PROGRAM P_AxisControl
VAR
END_VAR

//Axis Control program based on youtube series Twincat 3 NC Videos MB05a until MB17b plus MB22 by @electricalautomation https://www.youtube.com/watch?v=BxRAOdTks9I&list=PL762SfoJC-e8NbAUQ-H7a_TOdqrlBPCw4&index=25

AXIS1_LD();

GVL_AXIS1.bBC_ResetExe := G_Inputs.bJoystickLeftEnable OR G_Inputs.bAutoModeSelector;

GVL_AXIS1.EnuMoveVelDirection := G_Sensors.MCDirectionAxis1;

GVL_AXIS1.bBC_PowerEnCmd := G_Inputs.bManualModeSelector OR G_Inputs.bAutoModeSelector;
GVL_AXIS1.bBC_PowerEnNegative := G_Inputs.bManualModeSelector OR G_Inputs.bAutoModeSelector;
GVL_AXIS1.bBC_PowerEnPositive := G_Inputs.bManualModeSelector OR G_Inputs.bAutoModeSelector;

GVL_AXIS1.lrBC_JogVelocity := 100;
GVL_AXIS1.lrBC_PowerOverride := 50;

GVL_AXIS1.lrBC_MoveAbsPosition := GVL_InverseKinematics.fStrokeActuatorMainInverse*1000; //Position in mm

// Jog control

(*
IF G_Sensors.fJoystickLeftNormalizedX  > 0 AND G_Inputs.bJoystickLeftEnable THEN
	GVL_AXIS1.bBC_JogRev := TRUE;
ELSIF G_Sensors.fJoystickLeftNormalizedX < 0 AND G_Inputs.bJoystickLeftEnable THEN
	GVL_AXIS1.bBC_JogFwd := TRUE;
ELSE
	 GVL_AXIS1.bBC_JogFwd := FALSE;
	 GVL_AXIS1.bBC_JogRev := FALSE;
END_IF

*)



// Manual velocity control
IF G_Sensors.fJoystickLeftNormalizedX  > 0 AND G_Inputs.bJoystickLeftEnable AND G_Inputs.bManualModeSelector THEN
	GVL_AXIS1.lrBC_PowerOverride := ABS(G_Sensors.fJoystickLeftNormalizedX) * 100;
	GVL_AXIS1.stBC_VelCmd.EnuDirection := MC_Positive_Direction;
	GVL_AXIS1.stBC_VelCmd.bExe := TRUE;
ELSIF G_Sensors.fJoystickLeftNormalizedX < 0 AND G_Inputs.bJoystickLeftEnable AND G_Inputs.bManualModeSelector THEN
	GVL_AXIS1.lrBC_PowerOverride := ABS(G_Sensors.fJoystickLeftNormalizedX) * 100;
	GVL_AXIS1.stBC_VelCmd.EnuDirection := MC_Negative_Direction;
	GVL_AXIS1.stBC_VelCmd.bExe := TRUE;
ELSIF G_Inputs.bAutoModeSelector THEN
	GVL_AXIS1.lrBC_PowerOverride := 10;
	//GVL_AXIS1.stBC_VelCmd.EnuDirection := MC_Positive_Direction;
	GVL_AXIS1.stBC_VelCmd.bExe := TRUE;
	GVL_AXIS1.bBC_MoveAbsExe := TRUE;
ELSE
	 GVL_AXIS1.lrBC_PowerOverride := 0;
	 //GVL_AXIS1.stBC_VelCmd.EnuDirection := MC_Current_Direction;
	 GVL_AXIS1.stBC_VelCmd.bExe := FALSE;
END_IF


// Automatic position control

IF G_Inputs.bAutoModeSelector THEN
	GVL_AXIS1.lrBC_PowerOverride := 10;
	//GVL_AXIS1.stBC_VelCmd.EnuDirection := MC_Positive_Direction;
	GVL_AXIS1.stBC_VelCmd.bExe := TRUE;
	GVL_AXIS1.bBC_MoveAbsExe := TRUE;
ELSE
	 GVL_AXIS1.lrBC_PowerOverride := 0;
	 //GVL_AXIS1.stBC_VelCmd.EnuDirection := MC_Current_Direction;
	 GVL_AXIS1.stBC_VelCmd.bExe := FALSE;
END_IF


AXIS2_LD();

GVL_AXIS2.bSJ_ResetExe := G_Inputs.bJoystickRightEnable;

GVL_AXIS2.EnuMoveVelDirection := G_Sensors.MCDirectionAxis2;

GVL_AXIS2.bSJ_PowerEnCmd := G_Inputs.bManualModeSelector;
GVL_AXIS2.bSJ_PowerEnNegative := G_Inputs.bManualModeSelector;
GVL_AXIS2.bSJ_PowerEnPositive := G_Inputs.bManualModeSelector;

GVL_AXIS2.lrSJ_JogVelocity := 100;


// Velocity control
IF G_Sensors.fJoystickRightNormalizedX  > 0 AND G_Inputs.bJoystickRightEnable THEN
	GVL_AXIS2.lrSJ_PowerOverride := ABS(G_Sensors.fJoystickRightNormalizedX) * 100;
	GVL_AXIS2.stSJ_VelCmd.EnuDirection := MC_Positive_Direction;
	GVL_AXIS2.stSJ_VelCmd.bExe := TRUE;
ELSIF G_Sensors.fJoystickRightNormalizedX < 0 AND G_Inputs.bJoystickRightEnable THEN
	GVL_AXIS2.lrSJ_PowerOverride := ABS(G_Sensors.fJoystickRightNormalizedX) * 100;
	GVL_AXIS2.stSJ_VelCmd.EnuDirection := MC_Negative_Direction;
	GVL_AXIS2.stSJ_VelCmd.bExe := TRUE;
ELSE
	 GVL_AXIS2.lrSJ_PowerOverride := 0;
	 //GVL_AXIS2.stSJ_VelCmd.EnuDirection := MC_Current_Direction;
	 GVL_AXIS2.stSJ_VelCmd.bExe := FALSE;
END_IF


AXIS3_LD();

GVL_AXIS3.bTC_ResetExe := G_Inputs.bJoystickLeftEnable;

GVL_AXIS3.EnuMoveVelDirection := G_Sensors.MCDirectionAxis3;

GVL_AXIS3.bTC_PowerEnCmd := G_Inputs.bManualModeSelector;
GVL_AXIS3.bTC_PowerEnNegative := G_Inputs.bManualModeSelector;
GVL_AXIS3.bTC_PowerEnPositive := G_Inputs.bManualModeSelector;

GVL_AXIS3.lrTC_JogVelocity := 100;


// Velocity control
IF G_Sensors.fJoystickLeftNormalizedY  > 0 AND G_Inputs.bJoystickLeftEnable THEN
	GVL_AXIS3.lrTC_PowerOverride := ABS(G_Sensors.fJoystickLeftNormalizedY) * 100;
	GVL_AXIS3.stTC_VelCmd.EnuDirection := MC_Positive_Direction;
	GVL_AXIS3.stTC_VelCmd.bExe := TRUE;
ELSIF G_Sensors.fJoystickLeftNormalizedY < 0 AND G_Inputs.bJoystickLeftEnable THEN
	GVL_AXIS3.lrTC_PowerOverride := ABS(G_Sensors.fJoystickLeftNormalizedY) * 100;
	GVL_AXIS3.stTC_VelCmd.EnuDirection := MC_Negative_Direction;
	GVL_AXIS3.stTC_VelCmd.bExe := TRUE;
ELSE
	 GVL_AXIS3.lrTC_PowerOverride := 0;
	 //GVL_AXIS3.stTC_VelCmd.EnuDirection := MC_Current_Direction;
	 GVL_AXIS3.stTC_VelCmd.bExe := FALSE;
END_IF

(*
AXIS4_LD();

//Safety
GVL_Safety_AXIS4.bSafetyRestart := GVL_AXIS4.bInAckSignal;
GVL_Safety_AXIS4.bErrorAck		:= GVL_AXIS4.bInAckSignal;
GVL_Safety_AXIS4.bSafetyRun		:= TRUE;

//
GVL_AXIS4.bWM_ResetExe := G_Inputs.bJoystickLeftEnable;

GVL_AXIS4.EnuMoveVelDirection := G_Sensors.MCDirectionAxis4;

GVL_AXIS4.bWM_PowerEnCmd := G_Inputs.bManualModeSelector;
GVL_AXIS4.bWM_PowerEnNegative := G_Inputs.bManualModeSelector;
GVL_AXIS4.bWM_PowerEnPositive := G_Inputs.bManualModeSelector;

GVL_AXIS4.lrWM_JogVelocity := 100;
//GVL_AXIS4.lrWM_PowerOverride := 50;


// Velocity control
IF G_Sensors.fJoystickLeftNormalizedY  > 0 AND G_Inputs.bJoystickLeftEnable THEN
	GVL_AXIS4.lrWM_PowerOverride := ABS(G_Sensors.fJoystickLeftNormalizedY) * 100;
	GVL_AXIS4.stWM_VelCmd.EnuDirection := MC_Positive_Direction;
	GVL_AXIS4.stWM_VelCmd.bExe := TRUE;
ELSIF G_Sensors.fJoystickLeftNormalizedY < 0 AND G_Inputs.bJoystickLeftEnable THEN
	GVL_AXIS4.lrWM_PowerOverride := ABS(G_Sensors.fJoystickLeftNormalizedY) * 100;
	GVL_AXIS4.stWM_VelCmd.EnuDirection := MC_Negative_Direction;
	GVL_AXIS4.stWM_VelCmd.bExe := TRUE;
ELSE
	 GVL_AXIS4.lrWM_PowerOverride := 0;
	 GVL_AXIS4.stWM_VelCmd.EnuDirection := MC_Current_Direction;
	 GVL_AXIS4.stWM_VelCmd.bExe := FALSE;
END_IF
*)

METHOD AXIS1_LD : BOOL
VAR_INPUT
END_VAR
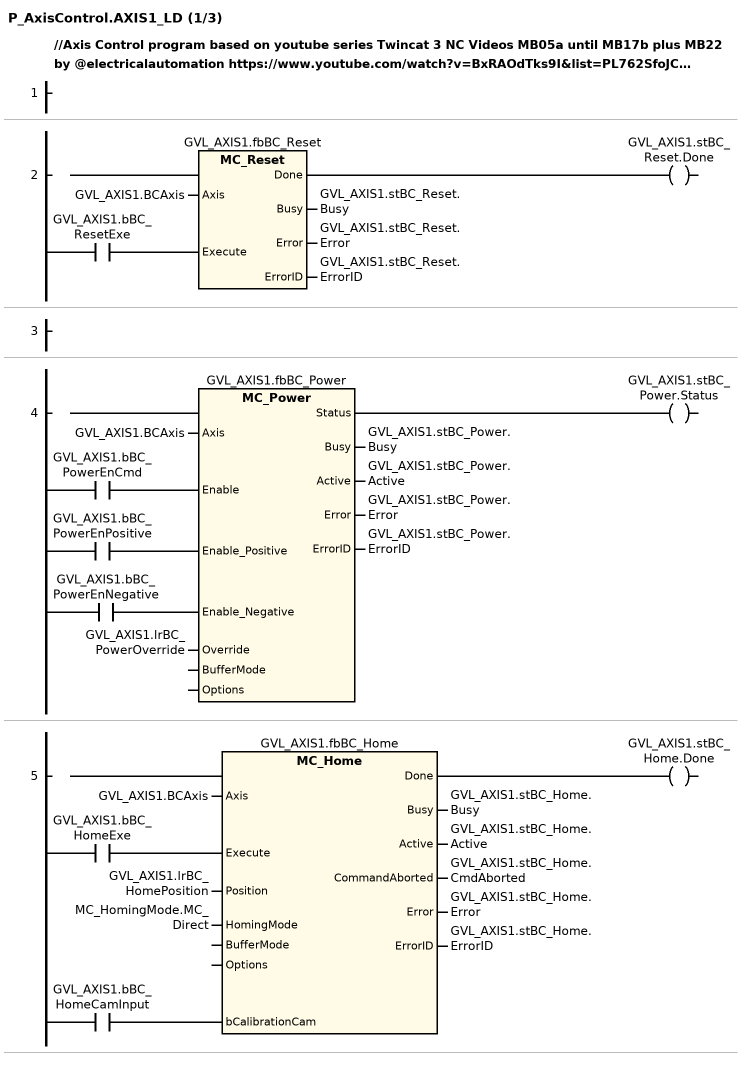
// NETWORK 1: //Axis Control program based on youtube series Twincat 3 NC Videos MB05a until MB17b plus MB22 by @electricalautomation https://www.youtube.com/watch?v=BxRAOdTks9I&list=PL762SfoJC-e8NbAUQ-H7a_TOdqrlBPCw4&index=25

// NETWORK 2
GVL_AXIS1.fbBC_Reset(
    Axis := GVL_AXIS1.BCAxis,
    Execute := GVL_AXIS1.bBC_ResetExe,
    Busy => GVL_AXIS1.stBC_Reset.Busy,
    Error => GVL_AXIS1.stBC_Reset.Error,
    ErrorID => GVL_AXIS1.stBC_Reset.ErrorID); // MC_Reset
GVL_AXIS1.stBC_Reset.Done := GVL_AXIS1.fbBC_Reset.Done;

// NETWORK 3

// NETWORK 4
GVL_AXIS1.fbBC_Power(
    Axis := GVL_AXIS1.BCAxis,
    Enable := GVL_AXIS1.bBC_PowerEnCmd,
    Enable_Positive := GVL_AXIS1.bBC_PowerEnPositive,
    Enable_Negative := GVL_AXIS1.bBC_PowerEnNegative,
    Override := GVL_AXIS1.lrBC_PowerOverride,
    Busy => GVL_AXIS1.stBC_Power.Busy,
    Active => GVL_AXIS1.stBC_Power.Active,
    Error => GVL_AXIS1.stBC_Power.Error,
    ErrorID => GVL_AXIS1.stBC_Power.ErrorID); // MC_Power
GVL_AXIS1.stBC_Power.Status := GVL_AXIS1.fbBC_Power.Status;

// NETWORK 5
GVL_AXIS1.fbBC_Home(
    Axis := GVL_AXIS1.BCAxis,
    Execute := GVL_AXIS1.bBC_HomeExe,
    Position := GVL_AXIS1.lrBC_HomePosition,
    HomingMode := MC_HomingMode.MC_Direct,
    bCalibrationCam := GVL_AXIS1.bBC_HomeCamInput,
    Busy => GVL_AXIS1.stBC_Home.Busy,
    Active => GVL_AXIS1.stBC_Home.Active,
    CommandAborted => GVL_AXIS1.stBC_Home.CmdAborted,
    Error => GVL_AXIS1.stBC_Home.Error,
    ErrorID => GVL_AXIS1.stBC_Home.ErrorID); // MC_Home
GVL_AXIS1.stBC_Home.Done := GVL_AXIS1.fbBC_Home.Done;

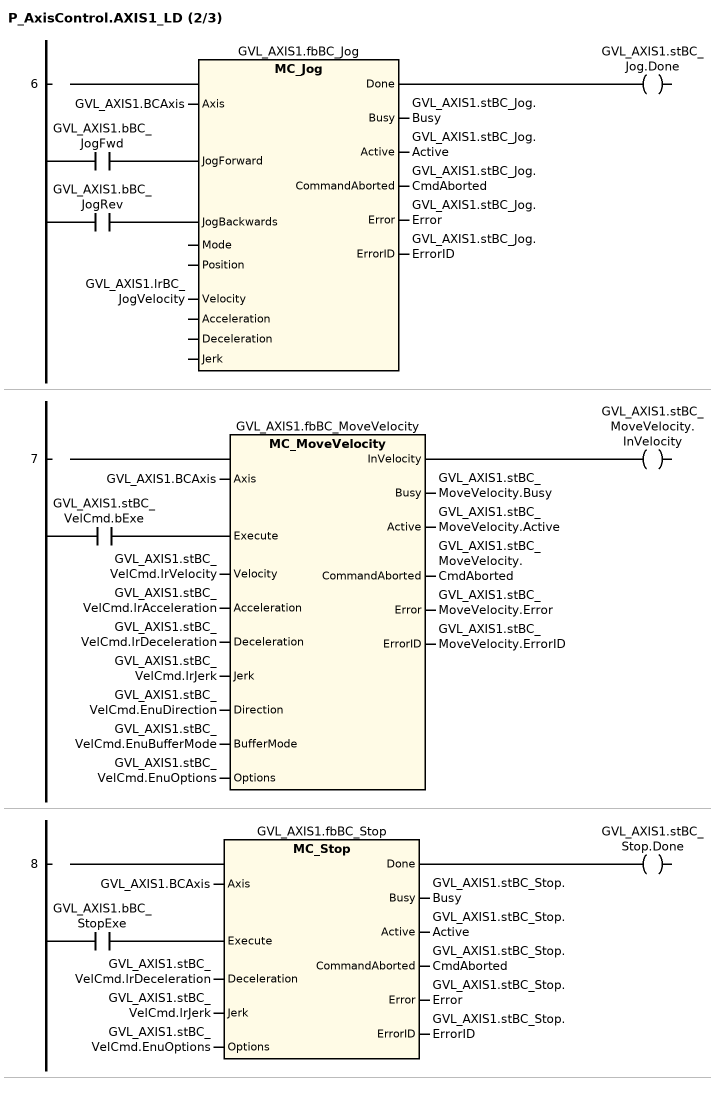
// NETWORK 6
GVL_AXIS1.fbBC_Jog(
    Axis := GVL_AXIS1.BCAxis,
    JogForward := GVL_AXIS1.bBC_JogFwd,
    JogBackwards := GVL_AXIS1.bBC_JogRev,
    Velocity := GVL_AXIS1.lrBC_JogVelocity,
    Busy => GVL_AXIS1.stBC_Jog.Busy,
    Active => GVL_AXIS1.stBC_Jog.Active,
    CommandAborted => GVL_AXIS1.stBC_Jog.CmdAborted,
    Error => GVL_AXIS1.stBC_Jog.Error,
    ErrorID => GVL_AXIS1.stBC_Jog.ErrorID); // MC_Jog
GVL_AXIS1.stBC_Jog.Done := GVL_AXIS1.fbBC_Jog.Done;

// NETWORK 7
GVL_AXIS1.fbBC_MoveVelocity(
    Axis := GVL_AXIS1.BCAxis,
    Execute := GVL_AXIS1.stBC_VelCmd.bExe,
    Velocity := GVL_AXIS1.stBC_VelCmd.lrVelocity,
    Acceleration := GVL_AXIS1.stBC_VelCmd.lrAcceleration,
    Deceleration := GVL_AXIS1.stBC_VelCmd.lrDeceleration,
    Jerk := GVL_AXIS1.stBC_VelCmd.lrJerk,
    Direction := GVL_AXIS1.stBC_VelCmd.EnuDirection,
    BufferMode := GVL_AXIS1.stBC_VelCmd.EnuBufferMode,
    Options := GVL_AXIS1.stBC_VelCmd.EnuOptions,
    Busy => GVL_AXIS1.stBC_MoveVelocity.Busy,
    Active => GVL_AXIS1.stBC_MoveVelocity.Active,
    CommandAborted => GVL_AXIS1.stBC_MoveVelocity.CmdAborted,
    Error => GVL_AXIS1.stBC_MoveVelocity.Error,
    ErrorID => GVL_AXIS1.stBC_MoveVelocity.ErrorID); // MC_MoveVelocity
GVL_AXIS1.stBC_MoveVelocity.InVelocity := GVL_AXIS1.fbBC_MoveVelocity.InVelocity;

// NETWORK 8
GVL_AXIS1.fbBC_Stop(
    Axis := GVL_AXIS1.BCAxis,
    Execute := GVL_AXIS1.bBC_StopExe,
    Deceleration := GVL_AXIS1.stBC_VelCmd.lrDeceleration,
    Jerk := GVL_AXIS1.stBC_VelCmd.lrJerk,
    Options := GVL_AXIS1.stBC_VelCmd.EnuOptions,
    Busy => GVL_AXIS1.stBC_Stop.Busy,
    Active => GVL_AXIS1.stBC_Stop.Active,
    CommandAborted => GVL_AXIS1.stBC_Stop.CmdAborted,
    Error => GVL_AXIS1.stBC_Stop.Error,
    ErrorID => GVL_AXIS1.stBC_Stop.ErrorID); // MC_Stop
GVL_AXIS1.stBC_Stop.Done := GVL_AXIS1.fbBC_Stop.Done;

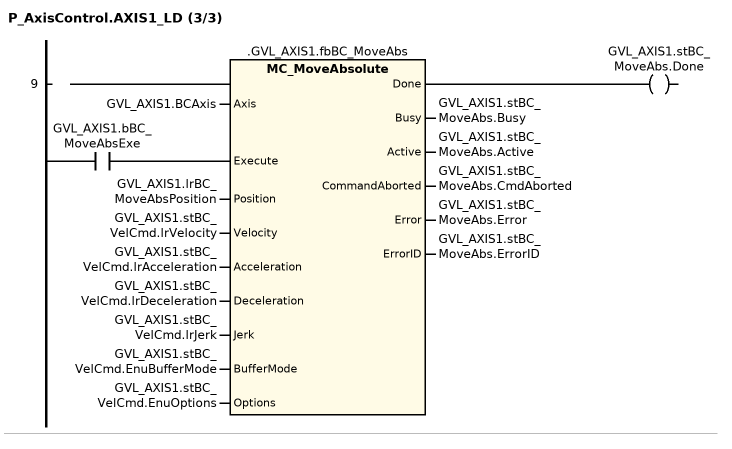
// NETWORK 9
.GVL_AXIS1.fbBC_MoveAbs(
    Axis := GVL_AXIS1.BCAxis,
    Execute := GVL_AXIS1.bBC_MoveAbsExe,
    Position := GVL_AXIS1.lrBC_MoveAbsPosition,
    Velocity := GVL_AXIS1.stBC_VelCmd.lrVelocity,
    Acceleration := GVL_AXIS1.stBC_VelCmd.lrAcceleration,
    Deceleration := GVL_AXIS1.stBC_VelCmd.lrDeceleration,
    Jerk := GVL_AXIS1.stBC_VelCmd.lrJerk,
    BufferMode := GVL_AXIS1.stBC_VelCmd.EnuBufferMode,
    Options := GVL_AXIS1.stBC_VelCmd.EnuOptions,
    Busy => GVL_AXIS1.stBC_MoveAbs.Busy,
    Active => GVL_AXIS1.stBC_MoveAbs.Active,
    CommandAborted => GVL_AXIS1.stBC_MoveAbs.CmdAborted,
    Error => GVL_AXIS1.stBC_MoveAbs.Error,
    ErrorID => GVL_AXIS1.stBC_MoveAbs.ErrorID); // MC_MoveAbsolute
GVL_AXIS1.stBC_MoveAbs.Done := .GVL_AXIS1.fbBC_MoveAbs.Done;
END_METHOD

METHOD AXIS2_LD : BOOL
VAR_INPUT
END_VAR
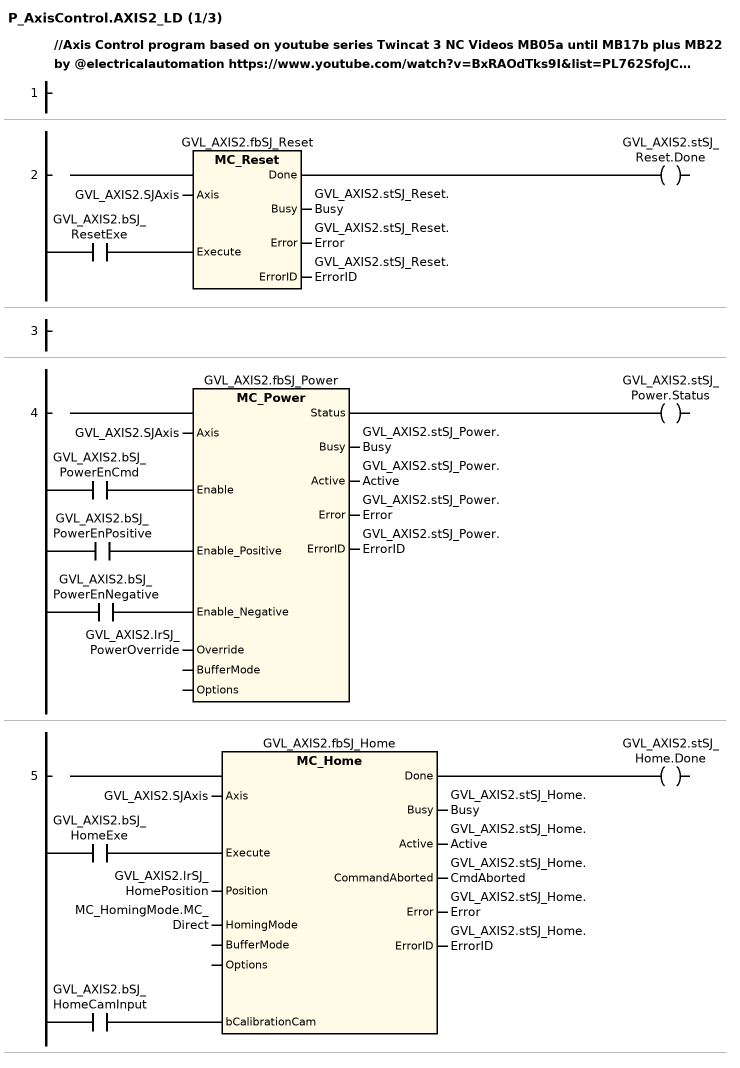
// NETWORK 1: //Axis Control program based on youtube series Twincat 3 NC Videos MB05a until MB17b plus MB22 by @electricalautomation https://www.youtube.com/watch?v=BxRAOdTks9I&list=PL762SfoJC-e8NbAUQ-H7a_TOdqrlBPCw4&index=25

// NETWORK 2
GVL_AXIS2.fbSJ_Reset(
    Axis := GVL_AXIS2.SJAxis,
    Execute := GVL_AXIS2.bSJ_ResetExe,
    Busy => GVL_AXIS2.stSJ_Reset.Busy,
    Error => GVL_AXIS2.stSJ_Reset.Error,
    ErrorID => GVL_AXIS2.stSJ_Reset.ErrorID); // MC_Reset
GVL_AXIS2.stSJ_Reset.Done := GVL_AXIS2.fbSJ_Reset.Done;

// NETWORK 3

// NETWORK 4
GVL_AXIS2.fbSJ_Power(
    Axis := GVL_AXIS2.SJAxis,
    Enable := GVL_AXIS2.bSJ_PowerEnCmd,
    Enable_Positive := GVL_AXIS2.bSJ_PowerEnPositive,
    Enable_Negative := GVL_AXIS2.bSJ_PowerEnNegative,
    Override := GVL_AXIS2.lrSJ_PowerOverride,
    Busy => GVL_AXIS2.stSJ_Power.Busy,
    Active => GVL_AXIS2.stSJ_Power.Active,
    Error => GVL_AXIS2.stSJ_Power.Error,
    ErrorID => GVL_AXIS2.stSJ_Power.ErrorID); // MC_Power
GVL_AXIS2.stSJ_Power.Status := GVL_AXIS2.fbSJ_Power.Status;

// NETWORK 5
GVL_AXIS2.fbSJ_Home(
    Axis := GVL_AXIS2.SJAxis,
    Execute := GVL_AXIS2.bSJ_HomeExe,
    Position := GVL_AXIS2.lrSJ_HomePosition,
    HomingMode := MC_HomingMode.MC_Direct,
    bCalibrationCam := GVL_AXIS2.bSJ_HomeCamInput,
    Busy => GVL_AXIS2.stSJ_Home.Busy,
    Active => GVL_AXIS2.stSJ_Home.Active,
    CommandAborted => GVL_AXIS2.stSJ_Home.CmdAborted,
    Error => GVL_AXIS2.stSJ_Home.Error,
    ErrorID => GVL_AXIS2.stSJ_Home.ErrorID); // MC_Home
GVL_AXIS2.stSJ_Home.Done := GVL_AXIS2.fbSJ_Home.Done;

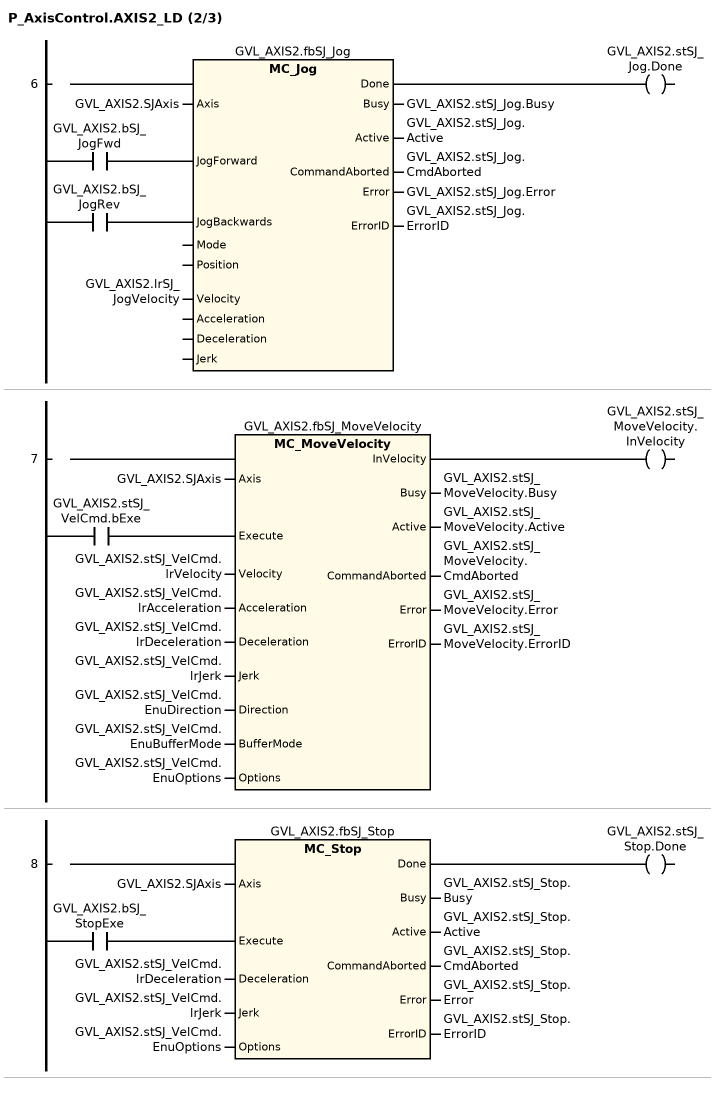
// NETWORK 6
GVL_AXIS2.fbSJ_Jog(
    Axis := GVL_AXIS2.SJAxis,
    JogForward := GVL_AXIS2.bSJ_JogFwd,
    JogBackwards := GVL_AXIS2.bSJ_JogRev,
    Velocity := GVL_AXIS2.lrSJ_JogVelocity,
    Busy => GVL_AXIS2.stSJ_Jog.Busy,
    Active => GVL_AXIS2.stSJ_Jog.Active,
    CommandAborted => GVL_AXIS2.stSJ_Jog.CmdAborted,
    Error => GVL_AXIS2.stSJ_Jog.Error,
    ErrorID => GVL_AXIS2.stSJ_Jog.ErrorID); // MC_Jog
GVL_AXIS2.stSJ_Jog.Done := GVL_AXIS2.fbSJ_Jog.Done;

// NETWORK 7
GVL_AXIS2.fbSJ_MoveVelocity(
    Axis := GVL_AXIS2.SJAxis,
    Execute := GVL_AXIS2.stSJ_VelCmd.bExe,
    Velocity := GVL_AXIS2.stSJ_VelCmd.lrVelocity,
    Acceleration := GVL_AXIS2.stSJ_VelCmd.lrAcceleration,
    Deceleration := GVL_AXIS2.stSJ_VelCmd.lrDeceleration,
    Jerk := GVL_AXIS2.stSJ_VelCmd.lrJerk,
    Direction := GVL_AXIS2.stSJ_VelCmd.EnuDirection,
    BufferMode := GVL_AXIS2.stSJ_VelCmd.EnuBufferMode,
    Options := GVL_AXIS2.stSJ_VelCmd.EnuOptions,
    Busy => GVL_AXIS2.stSJ_MoveVelocity.Busy,
    Active => GVL_AXIS2.stSJ_MoveVelocity.Active,
    CommandAborted => GVL_AXIS2.stSJ_MoveVelocity.CmdAborted,
    Error => GVL_AXIS2.stSJ_MoveVelocity.Error,
    ErrorID => GVL_AXIS2.stSJ_MoveVelocity.ErrorID); // MC_MoveVelocity
GVL_AXIS2.stSJ_MoveVelocity.InVelocity := GVL_AXIS2.fbSJ_MoveVelocity.InVelocity;

// NETWORK 8
GVL_AXIS2.fbSJ_Stop(
    Axis := GVL_AXIS2.SJAxis,
    Execute := GVL_AXIS2.bSJ_StopExe,
    Deceleration := GVL_AXIS2.stSJ_VelCmd.lrDeceleration,
    Jerk := GVL_AXIS2.stSJ_VelCmd.lrJerk,
    Options := GVL_AXIS2.stSJ_VelCmd.EnuOptions,
    Busy => GVL_AXIS2.stSJ_Stop.Busy,
    Active => GVL_AXIS2.stSJ_Stop.Active,
    CommandAborted => GVL_AXIS2.stSJ_Stop.CmdAborted,
    Error => GVL_AXIS2.stSJ_Stop.Error,
    ErrorID => GVL_AXIS2.stSJ_Stop.ErrorID); // MC_Stop
GVL_AXIS2.stSJ_Stop.Done := GVL_AXIS2.fbSJ_Stop.Done;

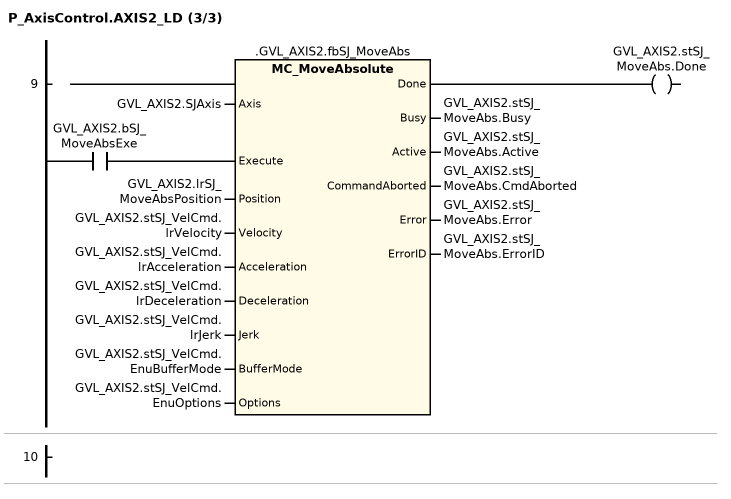
// NETWORK 9
.GVL_AXIS2.fbSJ_MoveAbs(
    Axis := GVL_AXIS2.SJAxis,
    Execute := GVL_AXIS2.bSJ_MoveAbsExe,
    Position := GVL_AXIS2.lrSJ_MoveAbsPosition,
    Velocity := GVL_AXIS2.stSJ_VelCmd.lrVelocity,
    Acceleration := GVL_AXIS2.stSJ_VelCmd.lrAcceleration,
    Deceleration := GVL_AXIS2.stSJ_VelCmd.lrDeceleration,
    Jerk := GVL_AXIS2.stSJ_VelCmd.lrJerk,
    BufferMode := GVL_AXIS2.stSJ_VelCmd.EnuBufferMode,
    Options := GVL_AXIS2.stSJ_VelCmd.EnuOptions,
    Busy => GVL_AXIS2.stSJ_MoveAbs.Busy,
    Active => GVL_AXIS2.stSJ_MoveAbs.Active,
    CommandAborted => GVL_AXIS2.stSJ_MoveAbs.CmdAborted,
    Error => GVL_AXIS2.stSJ_MoveAbs.Error,
    ErrorID => GVL_AXIS2.stSJ_MoveAbs.ErrorID); // MC_MoveAbsolute
GVL_AXIS2.stSJ_MoveAbs.Done := .GVL_AXIS2.fbSJ_MoveAbs.Done;

// NETWORK 10
END_METHOD

METHOD AXIS3_LD : BOOL
VAR_INPUT
END_VAR
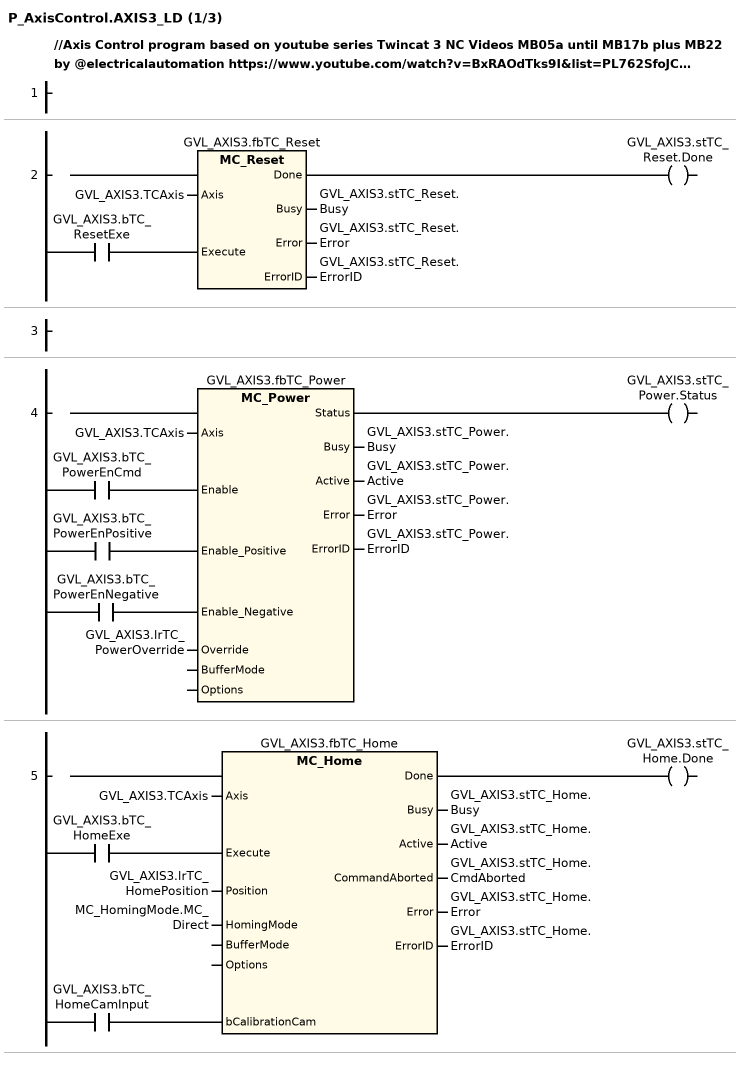
// NETWORK 1: //Axis Control program based on youtube series Twincat 3 NC Videos MB05a until MB17b plus MB22 by @electricalautomation https://www.youtube.com/watch?v=BxRAOdTks9I&list=PL762SfoJC-e8NbAUQ-H7a_TOdqrlBPCw4&index=25

// NETWORK 2
GVL_AXIS3.fbTC_Reset(
    Axis := GVL_AXIS3.TCAxis,
    Execute := GVL_AXIS3.bTC_ResetExe,
    Busy => GVL_AXIS3.stTC_Reset.Busy,
    Error => GVL_AXIS3.stTC_Reset.Error,
    ErrorID => GVL_AXIS3.stTC_Reset.ErrorID); // MC_Reset
GVL_AXIS3.stTC_Reset.Done := GVL_AXIS3.fbTC_Reset.Done;

// NETWORK 3

// NETWORK 4
GVL_AXIS3.fbTC_Power(
    Axis := GVL_AXIS3.TCAxis,
    Enable := GVL_AXIS3.bTC_PowerEnCmd,
    Enable_Positive := GVL_AXIS3.bTC_PowerEnPositive,
    Enable_Negative := GVL_AXIS3.bTC_PowerEnNegative,
    Override := GVL_AXIS3.lrTC_PowerOverride,
    Busy => GVL_AXIS3.stTC_Power.Busy,
    Active => GVL_AXIS3.stTC_Power.Active,
    Error => GVL_AXIS3.stTC_Power.Error,
    ErrorID => GVL_AXIS3.stTC_Power.ErrorID); // MC_Power
GVL_AXIS3.stTC_Power.Status := GVL_AXIS3.fbTC_Power.Status;

// NETWORK 5
GVL_AXIS3.fbTC_Home(
    Axis := GVL_AXIS3.TCAxis,
    Execute := GVL_AXIS3.bTC_HomeExe,
    Position := GVL_AXIS3.lrTC_HomePosition,
    HomingMode := MC_HomingMode.MC_Direct,
    bCalibrationCam := GVL_AXIS3.bTC_HomeCamInput,
    Busy => GVL_AXIS3.stTC_Home.Busy,
    Active => GVL_AXIS3.stTC_Home.Active,
    CommandAborted => GVL_AXIS3.stTC_Home.CmdAborted,
    Error => GVL_AXIS3.stTC_Home.Error,
    ErrorID => GVL_AXIS3.stTC_Home.ErrorID); // MC_Home
GVL_AXIS3.stTC_Home.Done := GVL_AXIS3.fbTC_Home.Done;

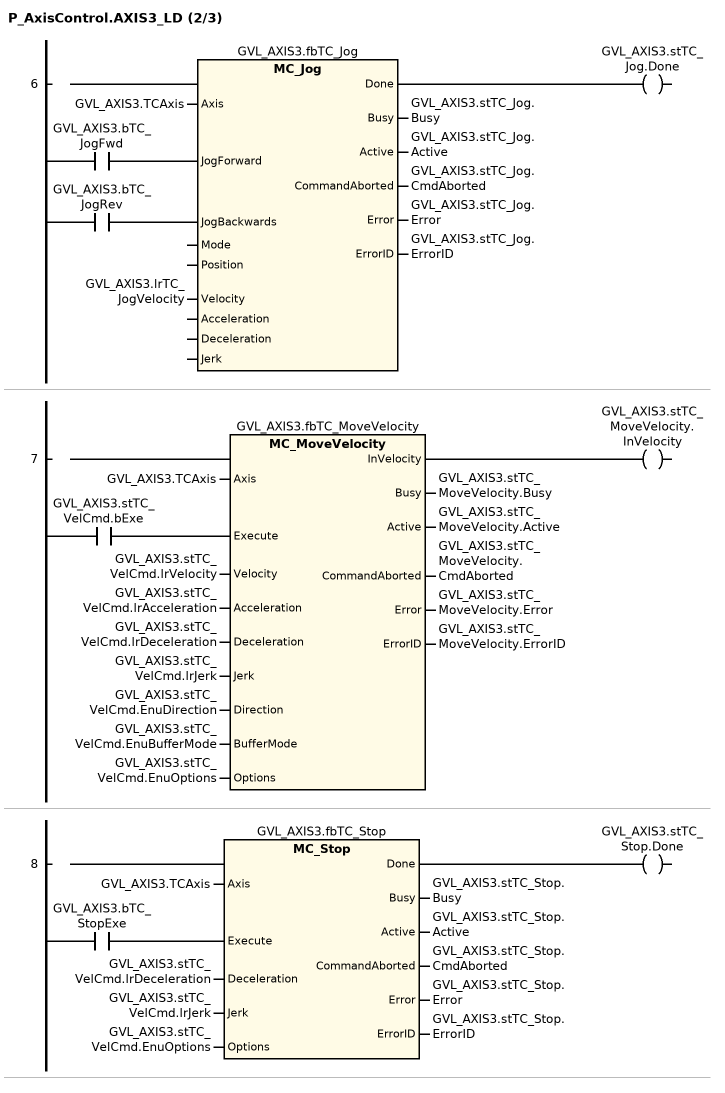
// NETWORK 6
GVL_AXIS3.fbTC_Jog(
    Axis := GVL_AXIS3.TCAxis,
    JogForward := GVL_AXIS3.bTC_JogFwd,
    JogBackwards := GVL_AXIS3.bTC_JogRev,
    Velocity := GVL_AXIS3.lrTC_JogVelocity,
    Busy => GVL_AXIS3.stTC_Jog.Busy,
    Active => GVL_AXIS3.stTC_Jog.Active,
    CommandAborted => GVL_AXIS3.stTC_Jog.CmdAborted,
    Error => GVL_AXIS3.stTC_Jog.Error,
    ErrorID => GVL_AXIS3.stTC_Jog.ErrorID); // MC_Jog
GVL_AXIS3.stTC_Jog.Done := GVL_AXIS3.fbTC_Jog.Done;

// NETWORK 7
GVL_AXIS3.fbTC_MoveVelocity(
    Axis := GVL_AXIS3.TCAxis,
    Execute := GVL_AXIS3.stTC_VelCmd.bExe,
    Velocity := GVL_AXIS3.stTC_VelCmd.lrVelocity,
    Acceleration := GVL_AXIS3.stTC_VelCmd.lrAcceleration,
    Deceleration := GVL_AXIS3.stTC_VelCmd.lrDeceleration,
    Jerk := GVL_AXIS3.stTC_VelCmd.lrJerk,
    Direction := GVL_AXIS3.stTC_VelCmd.EnuDirection,
    BufferMode := GVL_AXIS3.stTC_VelCmd.EnuBufferMode,
    Options := GVL_AXIS3.stTC_VelCmd.EnuOptions,
    Busy => GVL_AXIS3.stTC_MoveVelocity.Busy,
    Active => GVL_AXIS3.stTC_MoveVelocity.Active,
    CommandAborted => GVL_AXIS3.stTC_MoveVelocity.CmdAborted,
    Error => GVL_AXIS3.stTC_MoveVelocity.Error,
    ErrorID => GVL_AXIS3.stTC_MoveVelocity.ErrorID); // MC_MoveVelocity
GVL_AXIS3.stTC_MoveVelocity.InVelocity := GVL_AXIS3.fbTC_MoveVelocity.InVelocity;

// NETWORK 8
GVL_AXIS3.fbTC_Stop(
    Axis := GVL_AXIS3.TCAxis,
    Execute := GVL_AXIS3.bTC_StopExe,
    Deceleration := GVL_AXIS3.stTC_VelCmd.lrDeceleration,
    Jerk := GVL_AXIS3.stTC_VelCmd.lrJerk,
    Options := GVL_AXIS3.stTC_VelCmd.EnuOptions,
    Busy => GVL_AXIS3.stTC_Stop.Busy,
    Active => GVL_AXIS3.stTC_Stop.Active,
    CommandAborted => GVL_AXIS3.stTC_Stop.CmdAborted,
    Error => GVL_AXIS3.stTC_Stop.Error,
    ErrorID => GVL_AXIS3.stTC_Stop.ErrorID); // MC_Stop
GVL_AXIS3.stTC_Stop.Done := GVL_AXIS3.fbTC_Stop.Done;

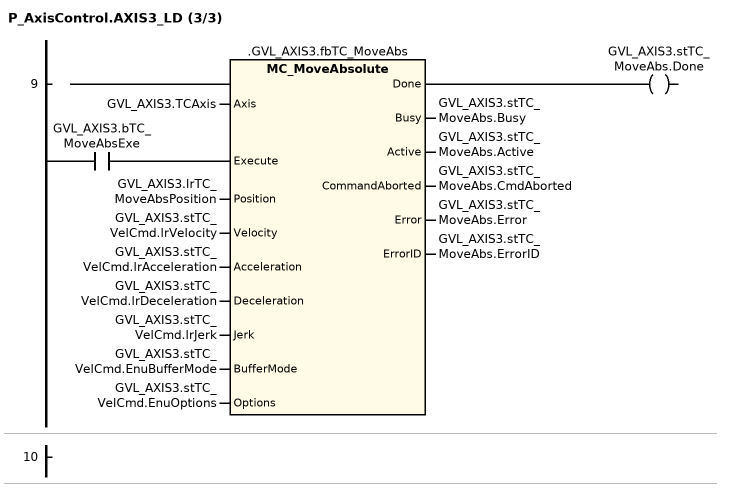
// NETWORK 9
.GVL_AXIS3.fbTC_MoveAbs(
    Axis := GVL_AXIS3.TCAxis,
    Execute := GVL_AXIS3.bTC_MoveAbsExe,
    Position := GVL_AXIS3.lrTC_MoveAbsPosition,
    Velocity := GVL_AXIS3.stTC_VelCmd.lrVelocity,
    Acceleration := GVL_AXIS3.stTC_VelCmd.lrAcceleration,
    Deceleration := GVL_AXIS3.stTC_VelCmd.lrDeceleration,
    Jerk := GVL_AXIS3.stTC_VelCmd.lrJerk,
    BufferMode := GVL_AXIS3.stTC_VelCmd.EnuBufferMode,
    Options := GVL_AXIS3.stTC_VelCmd.EnuOptions,
    Busy => GVL_AXIS3.stTC_MoveAbs.Busy,
    Active => GVL_AXIS3.stTC_MoveAbs.Active,
    CommandAborted => GVL_AXIS3.stTC_MoveAbs.CmdAborted,
    Error => GVL_AXIS3.stTC_MoveAbs.Error,
    ErrorID => GVL_AXIS3.stTC_MoveAbs.ErrorID); // MC_MoveAbsolute
GVL_AXIS3.stTC_MoveAbs.Done := .GVL_AXIS3.fbTC_MoveAbs.Done;

// NETWORK 10
END_METHOD

METHOD AXIS4_LD : BOOL
VAR_INPUT
END_VAR
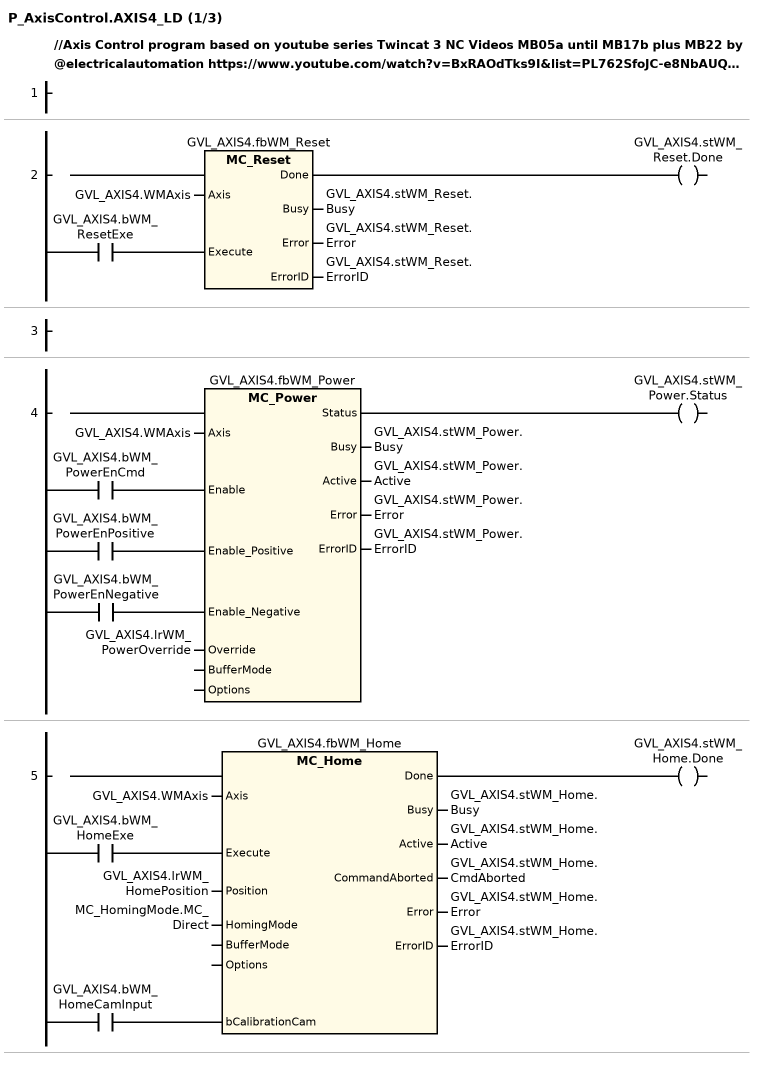
// NETWORK 1: //Axis Control program based on youtube series Twincat 3 NC Videos MB05a until MB17b plus MB22 by @electricalautomation https://www.youtube.com/watch?v=BxRAOdTks9I&list=PL762SfoJC-e8NbAUQ-H7a_TOdqrlBPCw4&index=25

// NETWORK 2
GVL_AXIS4.fbWM_Reset(
    Axis := GVL_AXIS4.WMAxis,
    Execute := GVL_AXIS4.bWM_ResetExe,
    Busy => GVL_AXIS4.stWM_Reset.Busy,
    Error => GVL_AXIS4.stWM_Reset.Error,
    ErrorID => GVL_AXIS4.stWM_Reset.ErrorID); // MC_Reset
GVL_AXIS4.stWM_Reset.Done := GVL_AXIS4.fbWM_Reset.Done;

// NETWORK 3

// NETWORK 4
GVL_AXIS4.fbWM_Power(
    Axis := GVL_AXIS4.WMAxis,
    Enable := GVL_AXIS4.bWM_PowerEnCmd,
    Enable_Positive := GVL_AXIS4.bWM_PowerEnPositive,
    Enable_Negative := GVL_AXIS4.bWM_PowerEnNegative,
    Override := GVL_AXIS4.lrWM_PowerOverride,
    Busy => GVL_AXIS4.stWM_Power.Busy,
    Active => GVL_AXIS4.stWM_Power.Active,
    Error => GVL_AXIS4.stWM_Power.Error,
    ErrorID => GVL_AXIS4.stWM_Power.ErrorID); // MC_Power
GVL_AXIS4.stWM_Power.Status := GVL_AXIS4.fbWM_Power.Status;

// NETWORK 5
GVL_AXIS4.fbWM_Home(
    Axis := GVL_AXIS4.WMAxis,
    Execute := GVL_AXIS4.bWM_HomeExe,
    Position := GVL_AXIS4.lrWM_HomePosition,
    HomingMode := MC_HomingMode.MC_Direct,
    bCalibrationCam := GVL_AXIS4.bWM_HomeCamInput,
    Busy => GVL_AXIS4.stWM_Home.Busy,
    Active => GVL_AXIS4.stWM_Home.Active,
    CommandAborted => GVL_AXIS4.stWM_Home.CmdAborted,
    Error => GVL_AXIS4.stWM_Home.Error,
    ErrorID => GVL_AXIS4.stWM_Home.ErrorID); // MC_Home
GVL_AXIS4.stWM_Home.Done := GVL_AXIS4.fbWM_Home.Done;

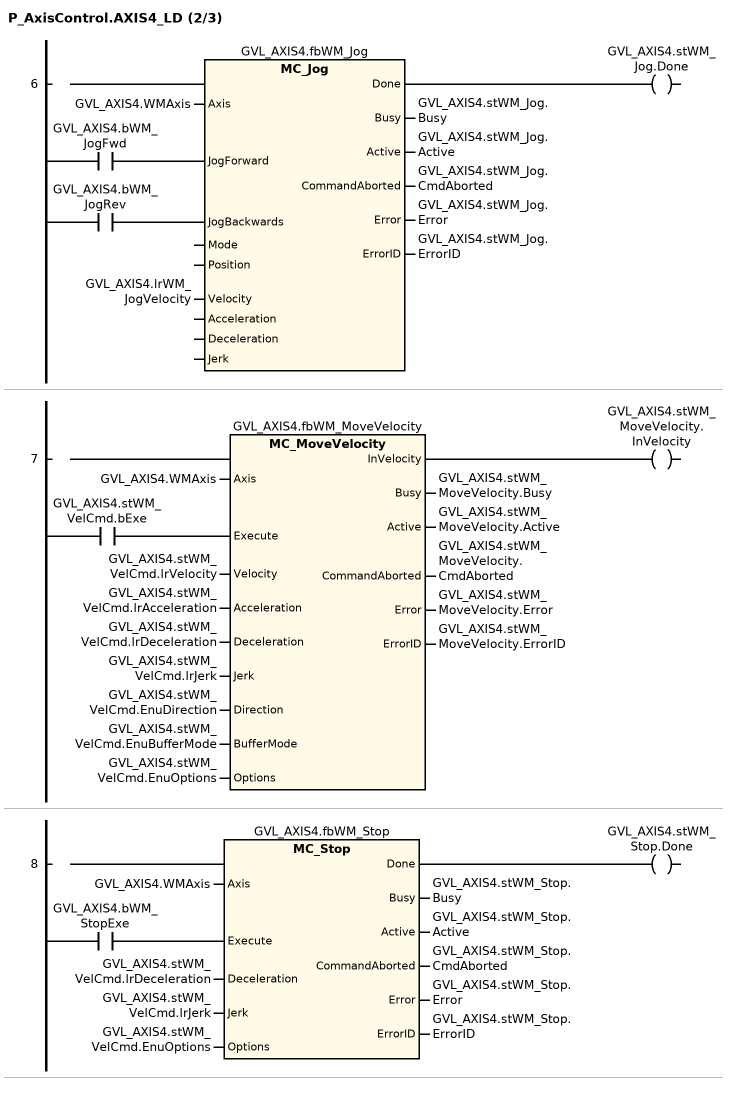
// NETWORK 6
GVL_AXIS4.fbWM_Jog(
    Axis := GVL_AXIS4.WMAxis,
    JogForward := GVL_AXIS4.bWM_JogFwd,
    JogBackwards := GVL_AXIS4.bWM_JogRev,
    Velocity := GVL_AXIS4.lrWM_JogVelocity,
    Busy => GVL_AXIS4.stWM_Jog.Busy,
    Active => GVL_AXIS4.stWM_Jog.Active,
    CommandAborted => GVL_AXIS4.stWM_Jog.CmdAborted,
    Error => GVL_AXIS4.stWM_Jog.Error,
    ErrorID => GVL_AXIS4.stWM_Jog.ErrorID); // MC_Jog
GVL_AXIS4.stWM_Jog.Done := GVL_AXIS4.fbWM_Jog.Done;

// NETWORK 7
GVL_AXIS4.fbWM_MoveVelocity(
    Axis := GVL_AXIS4.WMAxis,
    Execute := GVL_AXIS4.stWM_VelCmd.bExe,
    Velocity := GVL_AXIS4.stWM_VelCmd.lrVelocity,
    Acceleration := GVL_AXIS4.stWM_VelCmd.lrAcceleration,
    Deceleration := GVL_AXIS4.stWM_VelCmd.lrDeceleration,
    Jerk := GVL_AXIS4.stWM_VelCmd.lrJerk,
    Direction := GVL_AXIS4.stWM_VelCmd.EnuDirection,
    BufferMode := GVL_AXIS4.stWM_VelCmd.EnuBufferMode,
    Options := GVL_AXIS4.stWM_VelCmd.EnuOptions,
    Busy => GVL_AXIS4.stWM_MoveVelocity.Busy,
    Active => GVL_AXIS4.stWM_MoveVelocity.Active,
    CommandAborted => GVL_AXIS4.stWM_MoveVelocity.CmdAborted,
    Error => GVL_AXIS4.stWM_MoveVelocity.Error,
    ErrorID => GVL_AXIS4.stWM_MoveVelocity.ErrorID); // MC_MoveVelocity
GVL_AXIS4.stWM_MoveVelocity.InVelocity := GVL_AXIS4.fbWM_MoveVelocity.InVelocity;

// NETWORK 8
GVL_AXIS4.fbWM_Stop(
    Axis := GVL_AXIS4.WMAxis,
    Execute := GVL_AXIS4.bWM_StopExe,
    Deceleration := GVL_AXIS4.stWM_VelCmd.lrDeceleration,
    Jerk := GVL_AXIS4.stWM_VelCmd.lrJerk,
    Options := GVL_AXIS4.stWM_VelCmd.EnuOptions,
    Busy => GVL_AXIS4.stWM_Stop.Busy,
    Active => GVL_AXIS4.stWM_Stop.Active,
    CommandAborted => GVL_AXIS4.stWM_Stop.CmdAborted,
    Error => GVL_AXIS4.stWM_Stop.Error,
    ErrorID => GVL_AXIS4.stWM_Stop.ErrorID); // MC_Stop
GVL_AXIS4.stWM_Stop.Done := GVL_AXIS4.fbWM_Stop.Done;

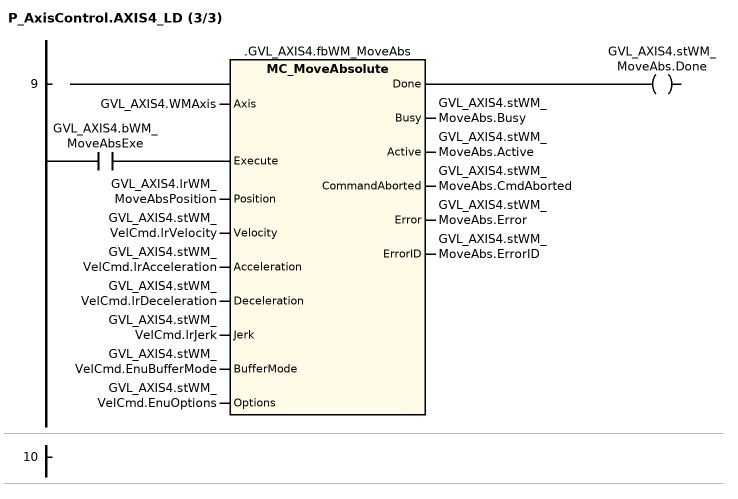
// NETWORK 9
.GVL_AXIS4.fbWM_MoveAbs(
    Axis := GVL_AXIS4.WMAxis,
    Execute := GVL_AXIS4.bWM_MoveAbsExe,
    Position := GVL_AXIS4.lrWM_MoveAbsPosition,
    Velocity := GVL_AXIS4.stWM_VelCmd.lrVelocity,
    Acceleration := GVL_AXIS4.stWM_VelCmd.lrAcceleration,
    Deceleration := GVL_AXIS4.stWM_VelCmd.lrDeceleration,
    Jerk := GVL_AXIS4.stWM_VelCmd.lrJerk,
    BufferMode := GVL_AXIS4.stWM_VelCmd.EnuBufferMode,
    Options := GVL_AXIS4.stWM_VelCmd.EnuOptions,
    Busy => GVL_AXIS4.stWM_MoveAbs.Busy,
    Active => GVL_AXIS4.stWM_MoveAbs.Active,
    CommandAborted => GVL_AXIS4.stWM_MoveAbs.CmdAborted,
    Error => GVL_AXIS4.stWM_MoveAbs.Error,
    ErrorID => GVL_AXIS4.stWM_MoveAbs.ErrorID); // MC_MoveAbsolute
GVL_AXIS4.stWM_MoveAbs.Done := .GVL_AXIS4.fbWM_MoveAbs.Done;

// NETWORK 10
END_METHOD

END_PROGRAM

(* stored: Version 1.1.0.1, ProductVersion 3.1.4024.12
   POU P_AxisControl: Id {5037aaa5-6389-4d48-9944-f1b3147b0b82}, SpecialFunc None
   Method AXIS1_LD: Id {a2ea73c2-d9a7-46bb-9d54-a37d5bff0a65}
   Method AXIS2_LD: Id {bdec519a-41ff-484d-9600-76653e24e62b}
   Method AXIS3_LD: Id {3773e93e-9c66-4353-b78a-0a74486d73ef}
   Method AXIS4_LD: Id {c68d9161-8577-4188-91d1-8d05a7c19713} *)
